PROGRAM MAIN
VAR
	
	PT1T2Parameter : PT1T2_Parameter_Strukt;	// Parameter des Prozesses
	PID_Parameter : PID_Parameter_Strukt;
	Modus : System_Modus_Enum := System_Modus_Enum.System_Init;
	T : REAL;
	PID_1 : PID_Regler;
	PT1T2_1 : PT1T2_Prozess;
	ref_rpm : REAL;
	conversion_rpm : EncoderOverflow_RPMConversion;
	y_rpm : REAL;
	u_volt : REAL;
	initial_voltage: REAL := 0;
END_VAR

T := 0.001;		// Abtastzeit 1ms
GVL_Real_Block.motor_enable := TRUE;


conversion_rpm(rpm_value => y_rpm);

// Systemparameter (PT1T2) definieren: Vollständig definiert
PT1T2_1.Param.K := 665;
PT1T2_1.Param.T_1 := 0.0073;		// Ti = 10 * T
PT1T2_1.Param.T_2 := 0.0513;		// Td = 0.1 * Ti

// Reglerparameter (PID)
PID_1.Param.K_p := 0.0026;//1/PT1T2_1.Param.K;		//Kp 1/K, 10/K, 100/K
PID_1.Param.T_i := 0.0386;//10 * T;
PID_1.Param.T_d := 0;//T;
PID_1.Param.u_max := 24;					// Von Stellgrössen Limitierung gegeben
PID_1.Param.u_min := -24;						// Von Stellgrössen Limitierung gegeben
PID_1.Param.ARW := TRUE;					// Ein-/Ausschaltung Anti-Reset Windup

// Regler für DC-Motor implementieren
PID_1(ref := ref_rpm, y := y_rpm, Modus := Modus, Param := PID_1.Param, T := T, u_r => u_volt);
GVL_Real_Block.motor_voltage := F_VOLTAGE_TO_INT(voltage := u_volt);

// A8 : Regelkreis implementieren
//PID_1(ref:= ref, y:= PT1T2_1.y_k, Modus := Modus, T := T);
//PT1T2_1(u := PID_1.u_r, Modus := Modus, T := T);

Modus := System_Modus_Enum.System_Run;


// 32767 fur +24 VDC und - 32767 fur -24VDC

END_PROGRAM

(* stored: Version 1.1.0.1, ProductVersion 3.1.4024.9
   POU MAIN: Id {bf7f390c-9673-4c1a-a757-c2e3b7e9acb8}, SpecialFunc None *)
